TYPE ST_MoverOptions :
STRUCT
	BaseMoveOptions	: REFERENCE TO Tc3_Mc3PlanarMotion.ST_MoveOnTrackOptions;
	TempGap : LREAL := stMoverConfig.TightMoverGap; //for ramping up/down gap over a sector
	OptionUpdateInterval : LREAL := 5.0; //mm
END_STRUCT
END_TYPE

(* stored: Version 1.1.0.1
   DUT ST_MoverOptions: Id {fde02a01-af06-0549-1846-c7bdbb2928d4} *)
